FUNCTION_BLOCK JSON_SERIALIZER (* Composite FB wrapping other FBs *)
  (* Standard: 61499-2 *)
  (* Version 1.0, 2023-04-20, valentinnodan *)
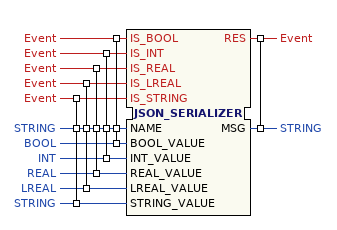
  EVENT_INPUT
    IS_BOOL WITH BOOL_VALUE, NAME; (* Normal Execution Request *)
    IS_INT WITH NAME, INT_VALUE;
    IS_REAL WITH NAME, REAL_VALUE;
    IS_LREAL WITH NAME, LREAL_VALUE;
    IS_STRING WITH NAME, STRING_VALUE;
  END_EVENT
  EVENT_OUTPUT
    RES WITH MSG; (* Execution Confirmation *)
  END_EVENT
  VAR_INPUT
    NAME : STRING;
    BOOL_VALUE : BOOL; (* Input event qualifier *)
    INT_VALUE : INT;
    REAL_VALUE : REAL;
    LREAL_VALUE : LREAL;
    STRING_VALUE : STRING;
  END_VAR
  VAR_OUTPUT
    MSG : STRING; (* Output event qualifier *)
  END_VAR
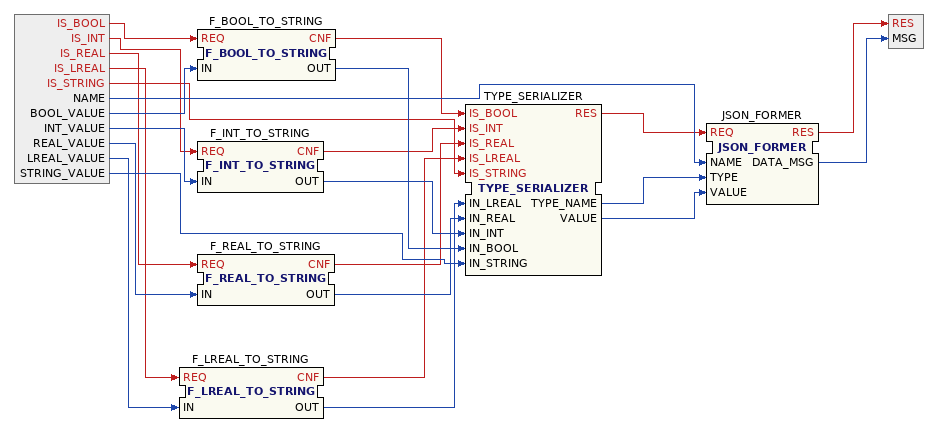
  FBS
    JSON_FORMER : JSON_FORMER;
    F_INT_TO_STRING : F_INT_TO_STRING;
    F_BOOL_TO_STRING : F_BOOL_TO_STRING;
    F_REAL_TO_STRING : F_REAL_TO_STRING;
    F_LREAL_TO_STRING : F_LREAL_TO_STRING;
    TYPE_SERIALIZER : TYPE_SERIALIZER;
  END_FBS
  EVENT_CONNECTIONS
    IS_BOOL TO F_BOOL_TO_STRING.REQ;
    IS_INT TO F_INT_TO_STRING.REQ;
    IS_REAL TO F_REAL_TO_STRING.REQ;
    IS_LREAL TO F_LREAL_TO_STRING.REQ;
    F_BOOL_TO_STRING.CNF TO TYPE_SERIALIZER.IS_BOOL;
    F_INT_TO_STRING.CNF TO TYPE_SERIALIZER.IS_INT;
    F_REAL_TO_STRING.CNF TO TYPE_SERIALIZER.IS_REAL;
    F_LREAL_TO_STRING.CNF TO TYPE_SERIALIZER.IS_LREAL;
    IS_STRING TO TYPE_SERIALIZER.IS_STRING;
    TYPE_SERIALIZER.RES TO JSON_FORMER.REQ;
    JSON_FORMER.RES TO RES;
  END_CONNECTIONS
  DATA_CONNECTIONS
    BOOL_VALUE TO F_BOOL_TO_STRING.IN;
    NAME TO JSON_FORMER.NAME;
    F_LREAL_TO_STRING.OUT TO TYPE_SERIALIZER.IN_LREAL;
    F_REAL_TO_STRING.OUT TO TYPE_SERIALIZER.IN_REAL;
    F_INT_TO_STRING.OUT TO TYPE_SERIALIZER.IN_INT;
    F_BOOL_TO_STRING.OUT TO TYPE_SERIALIZER.IN_BOOL;
    TYPE_SERIALIZER.TYPE_NAME TO JSON_FORMER.TYPE;
    TYPE_SERIALIZER.VALUE TO JSON_FORMER.VALUE;
    JSON_FORMER.DATA_MSG TO MSG;
    INT_VALUE TO F_INT_TO_STRING.IN;
    REAL_VALUE TO F_REAL_TO_STRING.IN;
    LREAL_VALUE TO F_LREAL_TO_STRING.IN;
    STRING_VALUE TO TYPE_SERIALIZER.IN_STRING;
  END_CONNECTIONS
END_FUNCTION_BLOCK
